FUNCTION F_UDINT_ARG : ST_Arg
VAR_INPUT
	nInput : UDINT;
END_VAR
VAR
	stArg : ST_Arg;
	sysVar_Info : __SYSTEM.VAR_INFO;
END_VAR

sysVar_Info := __VARINFO(nInput);
stArg.TypeClass := sysVar_Info.TypeClass;
stArg.pValue 	:= 0;
stArg.diSize 	:= SIZEOF(nInput);
stArg.sValue 	:= TO_STRING(nInput); 
F_UDINT_ARG := stArg;

END_FUNCTION

(* stored: Version 1.1.0.1, ProductVersion 3.1.4024.4
   POU F_UDINT_ARG: Id {6295efa5-b51c-4c22-b541-fb992b8dee52}, SpecialFunc None *)
